PROGRAM pouStation5
VAR
	stationMode: FB_Mode;
	tCalcNumberOfPages: REAL;
	ceil: REAL;
	PartBuild: FB_PartBuild;
	retvall: UDINT;
	// TODO
	tPartPresent: BOOL;
END_VAR

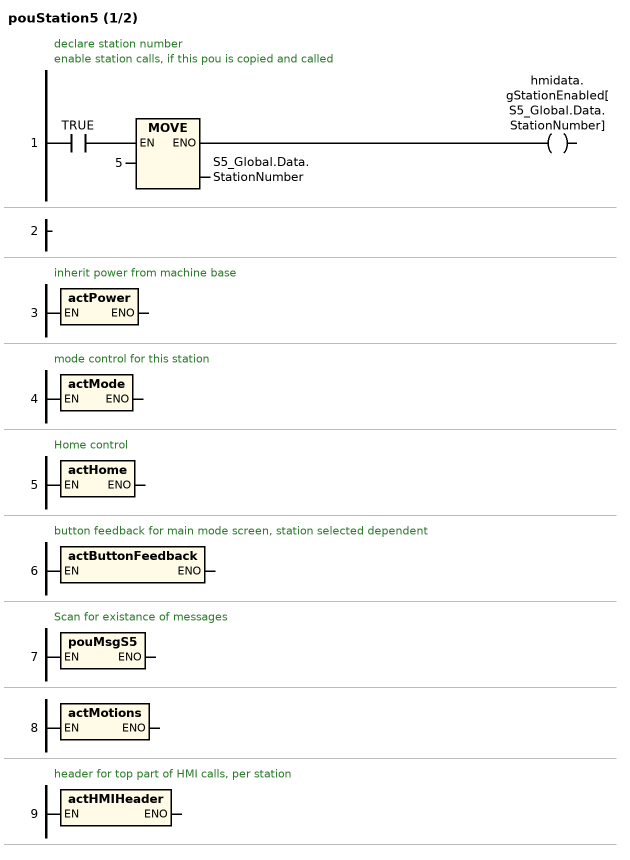
// NETWORK 1
// declare station number
// enable station calls, if this pou is copied and called
S5_Global.Data.StationNumber := 5;
hmidata.gStationEnabled[S5_Global.Data.StationNumber] := TRUE;

// NETWORK 2

// NETWORK 3
// inherit power from machine base
actPower();

// NETWORK 4
// mode control for this station
actMode();

// NETWORK 5
// Home control
actHome();

// NETWORK 6
// button feedback for main mode screen, station selected dependent
actButtonFeedback();

// NETWORK 7
// Scan for existance of messages
pouMsgS5();

// NETWORK 8
actMotions();

// NETWORK 9
// header for top part of HMI calls, per station
actHMIHeader();

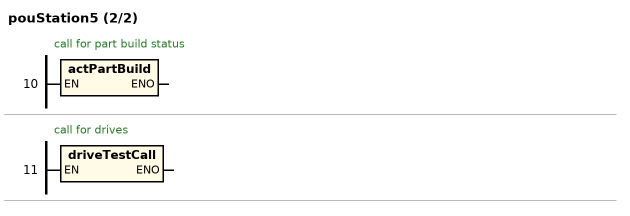
// NETWORK 10
// call for part build status
actPartBuild();

// NETWORK 11
// call for drives
driveTestCall();

ACTION actButtonFeedback:
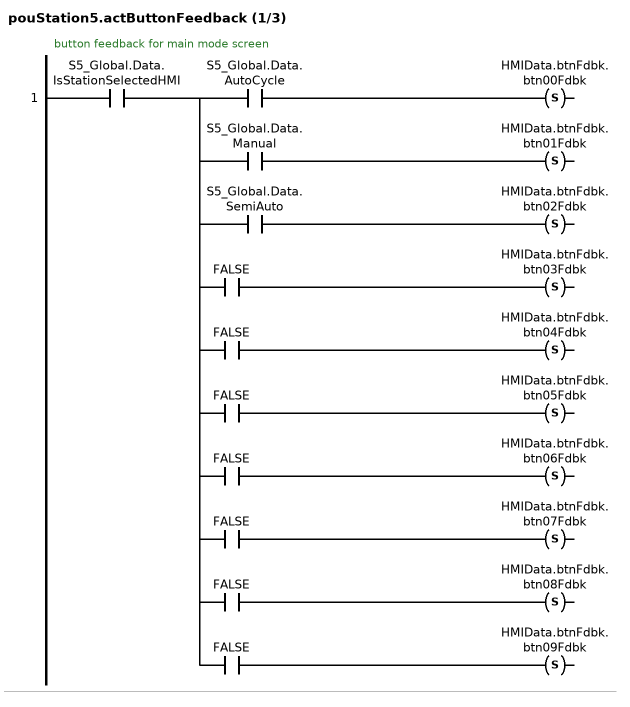
// NETWORK 1
// button feedback for main mode screen
HMIData.btnFdbk.btn00Fdbk S= S5_Global.Data.IsStationSelectedHMI AND S5_Global.Data.AutoCycle;
HMIData.btnFdbk.btn01Fdbk S= S5_Global.Data.IsStationSelectedHMI AND S5_Global.Data.Manual;
HMIData.btnFdbk.btn02Fdbk S= S5_Global.Data.IsStationSelectedHMI AND S5_Global.Data.SemiAuto;
HMIData.btnFdbk.btn03Fdbk S= S5_Global.Data.IsStationSelectedHMI AND FALSE;
HMIData.btnFdbk.btn04Fdbk S= S5_Global.Data.IsStationSelectedHMI AND FALSE;
HMIData.btnFdbk.btn05Fdbk S= S5_Global.Data.IsStationSelectedHMI AND FALSE;
HMIData.btnFdbk.btn06Fdbk S= S5_Global.Data.IsStationSelectedHMI AND FALSE;
HMIData.btnFdbk.btn07Fdbk S= S5_Global.Data.IsStationSelectedHMI AND FALSE;
HMIData.btnFdbk.btn08Fdbk S= S5_Global.Data.IsStationSelectedHMI AND FALSE;
HMIData.btnFdbk.btn09Fdbk S= S5_Global.Data.IsStationSelectedHMI AND FALSE;

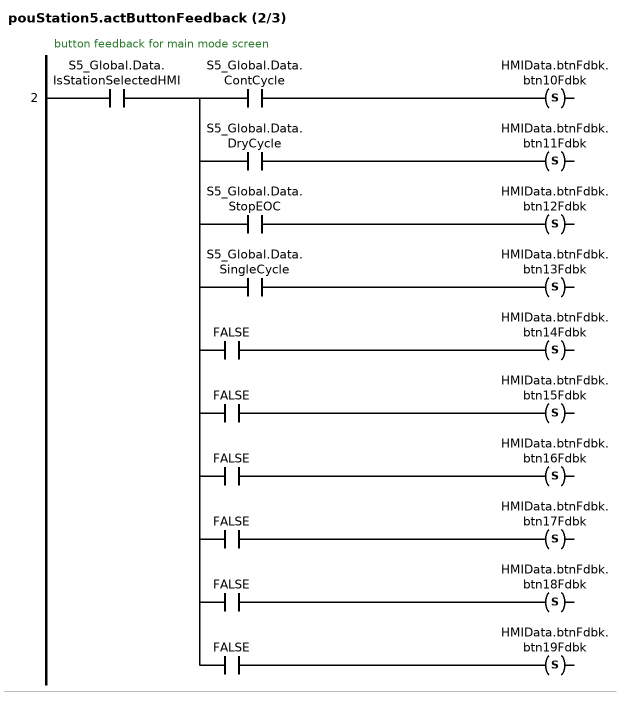
// NETWORK 2
// button feedback for main mode screen
HMIData.btnFdbk.btn10Fdbk S= S5_Global.Data.IsStationSelectedHMI AND S5_Global.Data.ContCycle;
HMIData.btnFdbk.btn11Fdbk S= S5_Global.Data.IsStationSelectedHMI AND S5_Global.Data.DryCycle;
HMIData.btnFdbk.btn12Fdbk S= S5_Global.Data.IsStationSelectedHMI AND S5_Global.Data.StopEOC;
HMIData.btnFdbk.btn13Fdbk S= S5_Global.Data.IsStationSelectedHMI AND S5_Global.Data.SingleCycle;
HMIData.btnFdbk.btn14Fdbk S= S5_Global.Data.IsStationSelectedHMI AND FALSE;
HMIData.btnFdbk.btn15Fdbk S= S5_Global.Data.IsStationSelectedHMI AND FALSE;
HMIData.btnFdbk.btn16Fdbk S= S5_Global.Data.IsStationSelectedHMI AND FALSE;
HMIData.btnFdbk.btn17Fdbk S= S5_Global.Data.IsStationSelectedHMI AND FALSE;
HMIData.btnFdbk.btn18Fdbk S= S5_Global.Data.IsStationSelectedHMI AND FALSE;
HMIData.btnFdbk.btn19Fdbk S= S5_Global.Data.IsStationSelectedHMI AND FALSE;

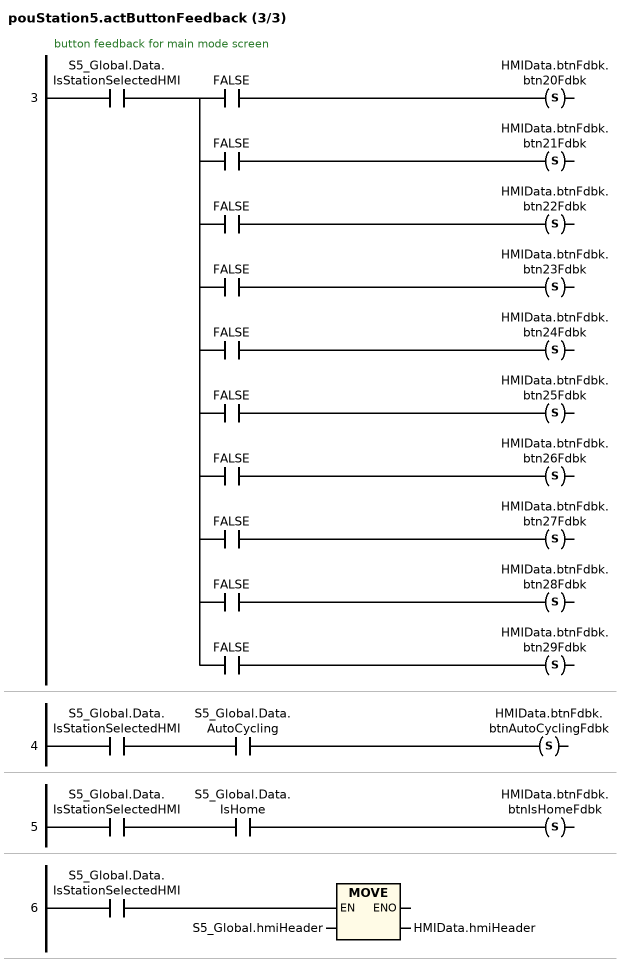
// NETWORK 3
// button feedback for main mode screen
HMIData.btnFdbk.btn20Fdbk S= S5_Global.Data.IsStationSelectedHMI AND FALSE;
HMIData.btnFdbk.btn21Fdbk S= S5_Global.Data.IsStationSelectedHMI AND FALSE;
HMIData.btnFdbk.btn22Fdbk S= S5_Global.Data.IsStationSelectedHMI AND FALSE;
HMIData.btnFdbk.btn23Fdbk S= S5_Global.Data.IsStationSelectedHMI AND FALSE;
HMIData.btnFdbk.btn24Fdbk S= S5_Global.Data.IsStationSelectedHMI AND FALSE;
HMIData.btnFdbk.btn25Fdbk S= S5_Global.Data.IsStationSelectedHMI AND FALSE;
HMIData.btnFdbk.btn26Fdbk S= S5_Global.Data.IsStationSelectedHMI AND FALSE;
HMIData.btnFdbk.btn27Fdbk S= S5_Global.Data.IsStationSelectedHMI AND FALSE;
HMIData.btnFdbk.btn28Fdbk S= S5_Global.Data.IsStationSelectedHMI AND FALSE;
HMIData.btnFdbk.btn29Fdbk S= S5_Global.Data.IsStationSelectedHMI AND FALSE;

// NETWORK 4
HMIData.btnFdbk.btnAutoCyclingFdbk S= S5_Global.Data.IsStationSelectedHMI AND S5_Global.Data.AutoCycling;

// NETWORK 5
HMIData.btnFdbk.btnIsHomeFdbk S= S5_Global.Data.IsStationSelectedHMI AND S5_Global.Data.IsHome;

// NETWORK 6
IF S5_Global.Data.IsStationSelectedHMI THEN HMIData.hmiHeader := S5_Global.hmiHeader; END_IF
END_ACTION

ACTION actHMIHeader:
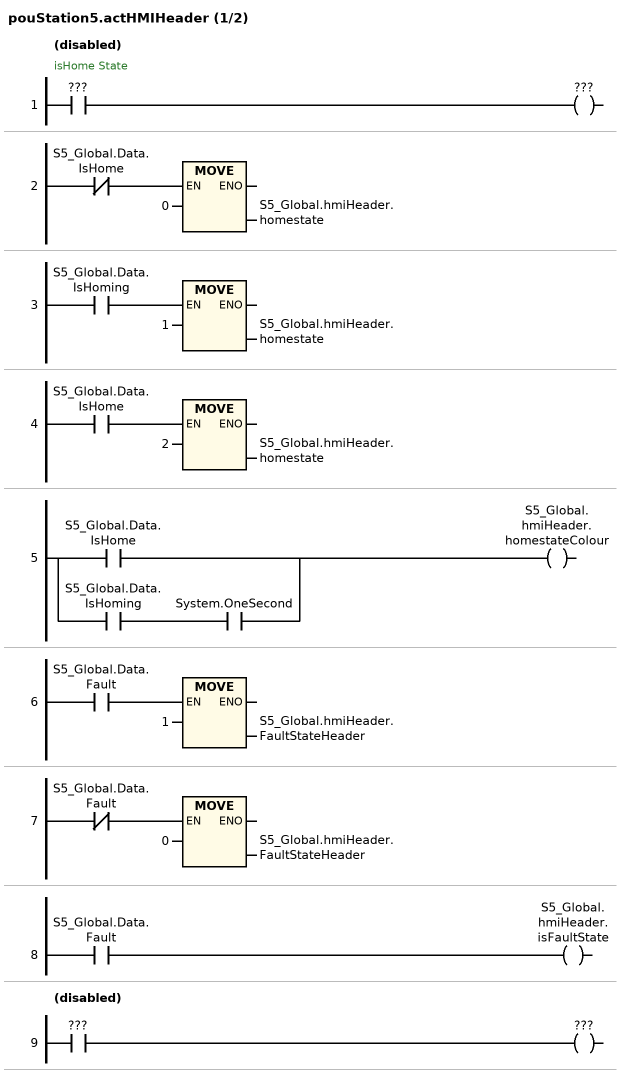
// NETWORK 1 (disabled)
// isHome State
// ??? := ???;

// NETWORK 2
IF NOT S5_Global.Data.IsHome THEN S5_Global.hmiHeader.homestate := 0; END_IF

// NETWORK 3
IF S5_Global.Data.IsHoming THEN S5_Global.hmiHeader.homestate := 1; END_IF

// NETWORK 4
IF S5_Global.Data.IsHome THEN S5_Global.hmiHeader.homestate := 2; END_IF

// NETWORK 5
S5_Global.hmiHeader.homestateColour := S5_Global.Data.IsHome OR S5_Global.Data.IsHoming AND System.OneSecond;

// NETWORK 6
IF S5_Global.Data.Fault THEN S5_Global.hmiHeader.FaultStateHeader := 1; END_IF

// NETWORK 7
IF NOT S5_Global.Data.Fault THEN S5_Global.hmiHeader.FaultStateHeader := 0; END_IF

// NETWORK 8
S5_Global.hmiHeader.isFaultState := S5_Global.Data.Fault;

// NETWORK 9 (disabled)
// ??? := ???;

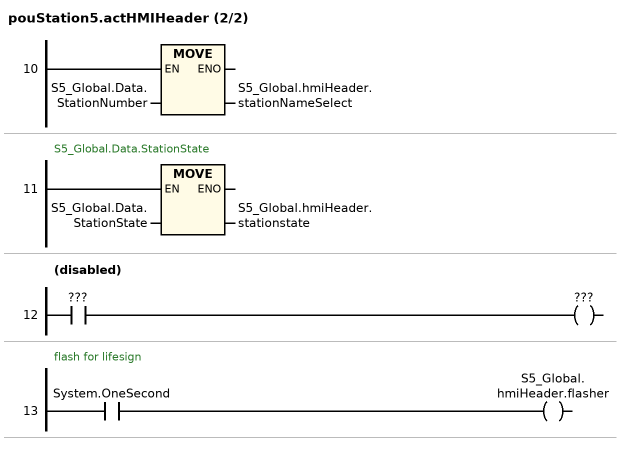
// NETWORK 10
S5_Global.hmiHeader.stationNameSelect := S5_Global.Data.StationNumber;

// NETWORK 11
// S5_Global.Data.StationState
S5_Global.hmiHeader.stationstate := S5_Global.Data.StationState;

// NETWORK 12 (disabled)
// ??? := ???;

// NETWORK 13
// flash for lifesign
S5_Global.hmiHeader.flasher := System.OneSecond;
END_ACTION

ACTION actHome:
//Set home status for station

IF 
//are all motions returned
S5_01_Motion_01_01.Motion.qReturnDepth AND
S5_01_Motion_01_02.Motion.qReturnDepth AND
S5_01_Motion_01_03.Motion.qReturnDepth AND
S5_01_Motion_01_04.Motion.qReturnDepth AND
S5_01_Motion_01_05.Motion.qReturnDepth AND
S5_01_Motion_01_06.Motion.qReturnDepth

	THEN
		//set IsHome value for station
		S5_Global.Data.IsHome := TRUE;
	ELSE
		S5_Global.Data.IsHome := FALSE;
END_IF
END_ACTION

ACTION actMaxNumStationPages:
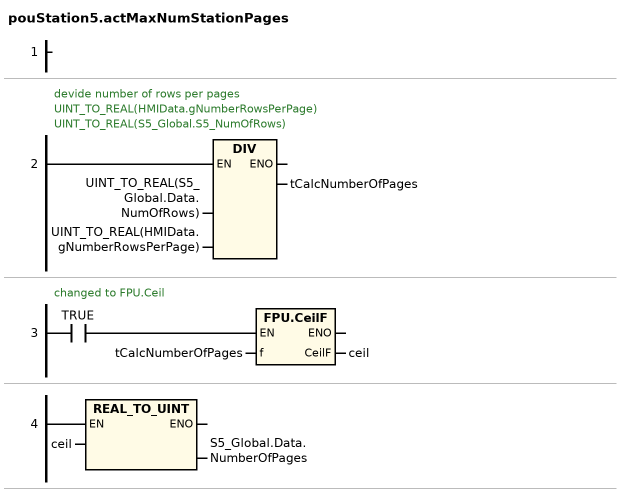
// NETWORK 1

// NETWORK 2
// devide number of rows per pages
// UINT_TO_REAL(HMIData.gNumberRowsPerPage)
// UINT_TO_REAL(S5_Global.S5_NumOfRows)
tCalcNumberOfPages := (UINT_TO_REAL(S5_Global.Data.NumOfRows)) / (UINT_TO_REAL(HMIData.gNumberRowsPerPage));

// NETWORK 3
// changed to FPU.Ceil
ceil := FPU.CeilF(f := tCalcNumberOfPages);

// NETWORK 4
S5_Global.Data.NumberOfPages := REAL_TO_UINT(ceil);
END_ACTION

ACTION actMode:
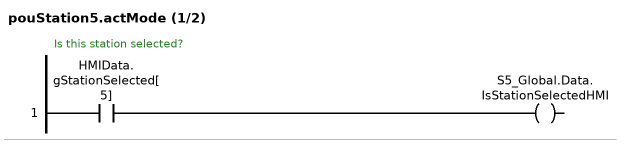
// NETWORK 1
// Is this station selected?
S5_Global.Data.IsStationSelectedHMI := HMIData.gStationSelected[5];

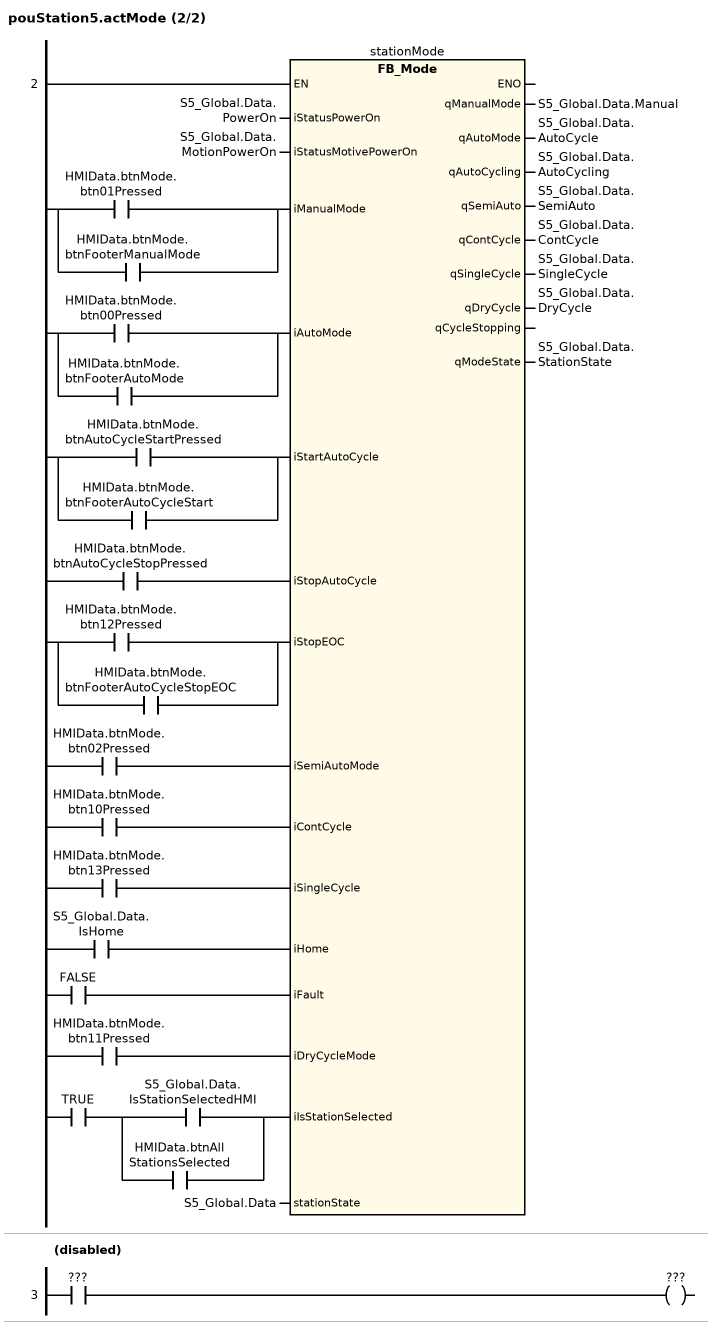
// NETWORK 2
stationMode(
    iStatusPowerOn := S5_Global.Data.PowerOn,
    iStatusMotivePowerOn := S5_Global.Data.MotionPowerOn,
    iManualMode := HMIData.btnMode.btn01Pressed OR HMIData.btnMode.btnFooterManualMode,
    iAutoMode := HMIData.btnMode.btn00Pressed OR HMIData.btnMode.btnFooterAutoMode,
    iStartAutoCycle := HMIData.btnMode.btnAutoCycleStartPressed OR HMIData.btnMode.btnFooterAutoCycleStart,
    iStopAutoCycle := HMIData.btnMode.btnAutoCycleStopPressed,
    iStopEOC := HMIData.btnMode.btn12Pressed OR HMIData.btnMode.btnFooterAutoCycleStopEOC,
    iSemiAutoMode := HMIData.btnMode.btn02Pressed,
    iContCycle := HMIData.btnMode.btn10Pressed,
    iSingleCycle := HMIData.btnMode.btn13Pressed,
    iHome := S5_Global.Data.IsHome,
    iFault := FALSE,
    iDryCycleMode := HMIData.btnMode.btn11Pressed,
    iIsStationSelected := TRUE AND (S5_Global.Data.IsStationSelectedHMI OR HMIData.btnAllStationsSelected),
    stationState := S5_Global.Data,
    qManualMode => S5_Global.Data.Manual,
    qAutoMode => S5_Global.Data.AutoCycle,
    qAutoCycling => S5_Global.Data.AutoCycling,
    qSemiAuto => S5_Global.Data.SemiAuto,
    qContCycle => S5_Global.Data.ContCycle,
    qSingleCycle => S5_Global.Data.SingleCycle,
    qDryCycle => S5_Global.Data.DryCycle,
    qModeState => S5_Global.Data.StationState); // FB_Mode

// NETWORK 3 (disabled)
// ??? := ???;
END_ACTION

ACTION actMotions:
//station 1 = 10000 index


//init number of rows
S5_Global.Data.NumOfRows := 0;

//page 1
S5_01_Motion_01_01();
S5_01_Motion_01_02();
S5_01_Motion_01_03();
S5_01_Motion_01_04();
S5_01_Motion_01_05();
S5_01_Motion_01_06();

//page 2
S5_01_Motion_02_07();
S5_01_Motion_02_08();
S5_01_Motion_02_09();
S5_01_Motion_02_10();
S5_01_Motion_02_11();
S5_01_Motion_02_12();

//page 3
S5_01_Motion_03_13();
S5_01_Motion_03_14();
S5_01_Motion_03_15();
S5_01_Motion_03_16();
S5_01_Motion_03_17();
S5_01_Motion_03_18();

//page 4
S5_01_Motion_04_19();
S5_01_Motion_04_20();
S5_01_Motion_04_21();
S5_01_Motion_04_22();
S5_01_Motion_04_23();
S5_01_Motion_04_24();

//page 5
S5_01_Motion_05_25();
S5_01_Motion_05_26();
S5_01_Motion_05_27();
S5_01_Motion_05_28();
S5_01_Motion_05_29();
S5_01_Motion_05_30();

//page 6
S5_01_Motion_06_31();
S5_01_Motion_06_32();
S5_01_Motion_06_33();
S5_01_Motion_06_34();
S5_01_Motion_06_35();
S5_01_Motion_06_36();

//must be called after motionRow calls
actMaxNumStationPages();
END_ACTION

ACTION actPartBuild:
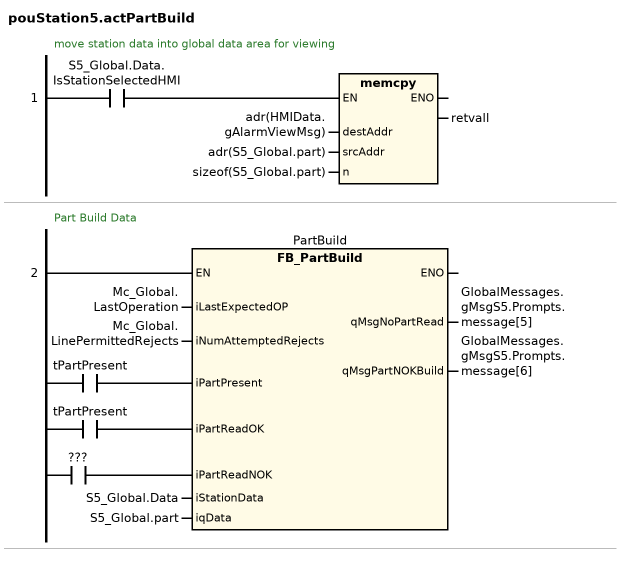
// NETWORK 1
// move station data into global data area for viewing
IF S5_Global.Data.IsStationSelectedHMI THEN
    retvall := memcpy(destAddr := adr(HMIData.gAlarmViewMsg), srcAddr := adr(S5_Global.part), n := sizeof(S5_Global.part));
END_IF

// NETWORK 2
// Part Build Data
PartBuild(
    iLastExpectedOP := Mc_Global.LastOperation,
    iNumAttemptedRejects := Mc_Global.LinePermittedRejects,
    iPartPresent := tPartPresent,
    iPartReadOK := tPartPresent,
    iStationData := S5_Global.Data,
    iqData := S5_Global.part,
    qMsgNoPartRead => GlobalMessages.gMsgS5.Prompts.message[5],
    qMsgPartNOKBuild => GlobalMessages.gMsgS5.Prompts.message[6]); // FB_PartBuild
END_ACTION

ACTION actPower:
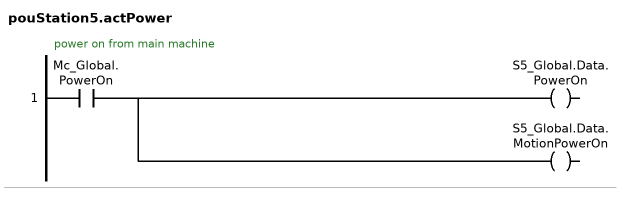
// NETWORK 1
// power on from main machine
S5_Global.Data.PowerOn := Mc_Global.PowerOn;
S5_Global.Data.MotionPowerOn := Mc_Global.PowerOn;
END_ACTION

END_PROGRAM

(* stored: Version 1.1.0.1, ProductVersion 3.1.4024.12
   POU pouStation5: Id {538ece2f-2153-4f20-9a3f-b8babb351419}, SpecialFunc None
   Action actButtonFeedback: Id {6ebd5c7e-77a6-4d8a-b67d-7624369e3e26}
   Action actHMIHeader: Id {1f0cbc1c-0b6c-4494-a071-979fb099cad0}
   Action actHome: Id {2fee892e-409b-48ea-ae00-80d81e1ad144}
   Action actMaxNumStationPages: Id {536d5900-6f46-464b-87e5-a43a2dd591c9}
   Action actMode: Id {4ee99afc-0968-4b20-914f-b9fabfbdd83c}
   Action actMotions: Id {7d95f8cf-d517-4089-90a7-0d014c628f52}
   Action actPartBuild: Id {b786c992-a10f-4627-ad0e-3b0047033ba0}
   Action actPower: Id {b903eb56-0e1e-4ab4-820e-70c0a498c463} *)
